// TIA Portal V17 export
// export: Created 2025-03-05T07:59:22.9336726Z, ExportSetting WithDefaults, DisplayName Totally Integrated Automation Portal, DisplayVersion V17 Update 8, DisplayName TIA Portal Openness, DisplayVersion V17 Update 8, DisplayName TIA Portal Version Control Interface, DisplayVersion V17, DisplayName SINAMICS Startdrive Advanced, DisplayVersion V17 SP2, DisplayName SINAMICS Startdrive G110M, G120, G120C, G120D, G120P, G115D, DisplayVersion V17 SP2, DisplayName SINAMICS Startdrive G130, G150, S120, S150, SINAMICS MV, S210, DisplayVersion V17 SP2, DisplayName STEP 7 Professional, DisplayVersion V17 Update 8, DisplayName SINUMERIK ONE STEP 7 Toolbox, DisplayVersion V17 Update 12, DisplayName SINUMERIK 840D sl STEP 7 Toolbox, DisplayVersion V17 Update 12, DisplayName STEP 7 Safety, DisplayVersion V17 Update 6, DisplayName WinCC Advanced, DisplayVersion V17 Update 8
DATA_BLOCK "DB7340_POWDER_PLC_INTERLOCK"   // DB7340
{ S7_Optimized_Access := 'FALSE'; DB_Accessible_From_OPC_UA := 'FALSE' }
AUTHOR : ETXETAR
VERSION : 1.0
// stored: AutoNumber false, DBAccessibleFromOPCUA false, DBAccessibleFromWebserver true, IsOnlyStoredInLoadMemory false, IsWriteProtectedInAS false
   VAR RETAIN
      POWDER_TO_NCU : Struct
         LIFE_BIT : Bool;   // LIFE BIT
         POWDER_UNIT_01_READY_TO_RUN : Bool;   // POWDER UNIT 01 READY TO RUN
         POWDER_UNIT_02_READY_TO_RUN : Bool;   // POWDER UNIT 02 READY TO RUN
         POWDER_UNIT_01_STOPPED : Bool;   // POWDER UNIT 01 STOPPED
         POWDER_UNIT_02_STOPPED : Bool;   // POWDER UNIT 02 STOPPED
         SPARE_05 : Bool;
         SPARE_06 : Bool;
         SPARE_07 : Bool;
         POWDER_PLC_AUTO_MODE : Bool;   // POWDER PLC IN AUTO MODE
         POWDER_PLC_MAN_MODE : Bool;   // POWDER PLC IN MANUAL MODE
         SPARE_12 : Bool;
         SPARE_13 : Bool;
         SPARE_14 : Bool;
         SPARE_15 : Bool;
         SPARE_16 : Bool;
         SPARE_17 : Bool;
         SWITCHED_ON_POWDER_UNIT_01 : Bool;   // SWITCHED ON POWDER UNIT 01
         SWITCHED_ON_POWDER_UNIT_02 : Bool;   // SWITCHED ON POWDER UNIT 02
         SWITCHED_OFF_POWDER_UNIT_01 : Bool;   // SWITCHED OFF POWDER UNIT 01
         SWITCHED_OFF_POWDER_UNIT_02 : Bool;   // SWITCHED OFF POWDER UNIT 02
         SWITCHED_ON_TEMPERATURE_JACKET_UNIT_01 : Bool;   // SWITCHED ON TEMPERATURE JACKET UNIT 01
         SWITCHED_ON_TEMPERATURE_JACKET_UNIT_02 : Bool;   // SWITCHED ON TEMPERATURE JACKET UNIT 02
         SWITCHED_OFF_TEMPERATURE_JACKET_UNIT_01 : Bool;   // SWITCHED OFF TEMPERATURE JACKET UNIT 01
         SWITCHED_OFF_TEMPERATURE_JACKET_UNIT_02 : Bool;   // SWITCHED OFF TEMPERATURE JACKET UNIT 02
         SPARE_30 : Bool;
         SPARE_31 : Bool;
         SPARE_32 : Bool;
         SPARE_33 : Bool;
         SPARE_34 : Bool;
         SPARE_35 : Bool;
         SPARE_36 : Bool;
         SPARE_37 : Bool;
         SPARE_38 : Bool;
         SPARE_39 : Bool;
         SPARE_40 : Bool;
         SPARE_41 : Bool;
         SPARE_44 : Bool;
         SPARE_45 : Bool;
         SPARE_46 : Bool;
         SPARE_47 : Bool;
         POWDER_UNIT_01_ALARM : Bool;   // POWDER UNIT 01 ALARM
         POWDER_UNIT_02_ALARM : Bool;   // POWDER UNIT 02 ALARM
         SPARE_52 : Bool;
         SPARE_53 : Bool;
         SPARE_54 : Bool;
         SPARE_55 : Bool;
         SPARE_56 : Bool;
         SPARE_57 : Bool;
         SPARE_60 : Bool;
         SPARE_61 : Bool;
         SPARE_62 : Bool;
         SPARE_63 : Bool;
         SPARE_64 : Bool;
         SPARE_65 : Bool;
         SPARE_66 : Bool;
         SPARE_67 : Bool;
         SPARE_70 : Bool;
         SPARE_71 : Bool;
         SPARE_72 : Bool;
         SPARE_73 : Bool;
         SPARE_74 : Bool;
         SPARE_75 : Bool;
         SPARE_76 : Bool;
         SPARE_77 : Bool;
         SPARE_80 : Bool;
         SPARE_81 : Bool;
         SPARE_82 : Bool;
         SPARE_83 : Bool;
         SPARE_84 : Bool;
         SPARE_85 : Bool;
         SPARE_86 : Bool;
         SPARE_87 : Bool;
         SPARE_90 : Bool;
         SPARE_91 : Bool;
         SPARE_92 : Bool;
         SPARE_93 : Bool;
         SPARE_94 : Bool;
         SPARE_95 : Bool;
         SPARE_96 : Bool;
         SPARE_97 : Bool;
         UNIT_01_POWDER_FEEDER_1_CARRIER_GAS_ACTUAL_LINE_1 : Real;   // UNIT 01 POWDER FEEDER 1 CARRIER GAS ACTUAL LINE 1
         UNIT_01_POWDER_FEEDER_1_CARRIER_GAS_ACTUAL_LINE_2 : Real;   // UNIT 01 POWDER FEEDER 1 CARRIER GAS ACTUAL LINE 2
         UNIT_01_POWDER_FEEDER_1_DISK_SPEED_ACTUAL_LINE_1 : Real;   // UNIT 01 POWDER FEEDER 1 DISK SPEED ACTUAL LINE 1
         UNIT_01_POWDER_FEEDER_1_DISK_SPEED_ACTUAL_LINE_2 : Real;   // UNIT 01 POWDER FEEDER 1 DISK SPEED ACTUAL LINE 2
         UNIT_01_POWDER_FEEDER_1_STIRRER_SPEED_ACTUAL_LINE_1 : Real;   // UNIT 01 POWDER FEEDER 1 STIRRER SPEED ACTUAL LINE 1
         UNIT_01_POWDER_FEEDER_1_STIRRER_SPEED_ACTUAL_LINE_2 : Real;   // UNIT 01 POWDER FEEDER 1 STIRRER SPEED ACTUAL LINE 2
         UNIT_01_POWDER_FEEDER_1_HOPPER_TEMPERATURE_ACTUAL_LINE_1 : Real;   // UNIT 01 POWDER FEEDER 1 HOPPER TEMPERATURE ACTUAL LINE 1
         UNIT_01_POWDER_FEEDER_1_HOPPER_TEMPERATURE_ACTUAL_LINE_2 : Real;   // UNIT 01 POWDER FEEDER 1 HOPPER TEMPERATURE ACTUAL LINE 2
         UNIT_02_POWDER_FEEDER_1_CARRIER_GAS_ACTUAL_LINE_1 : Real;   // UNIT 02 POWDER FEEDER 1 CARRIER GAS ACTUAL LINE 1
         UNIT_02_POWDER_FEEDER_1_CARRIER_GAS_ACTUAL_LINE_2 : Real;   // UNIT 02 POWDER FEEDER 1 CARRIER GAS ACTUAL LINE 2
         UNIT_02_POWDER_FEEDER_1_DISK_SPEED_ACTUAL_LINE_1 : Real;   // UNIT 02 POWDER FEEDER 1 DISK SPEED ACTUAL LINE 1
         UNIT_02_POWDER_FEEDER_1_DISK_SPEED_ACTUAL_LINE_2 : Real;   // UNIT 02 POWDER FEEDER 1 DISK SPEED ACTUAL LINE 2
         UNIT_02_POWDER_FEEDER_1_STIRRER_SPEED_ACTUAL_LINE_1 : Real;   // UNIT 02 POWDER FEEDER 1 STIRRER SPEED ACTUAL LINE 1
         UNIT_02_POWDER_FEEDER_1_STIRRER_SPEED_ACTUAL_LINE_2 : Real;   // UNIT 02 POWDER FEEDER 1 STIRRER SPEED ACTUAL LINE 2
         UNIT_02_POWDER_FEEDER_1_HOPPER_TEMPERATURE_ACTUAL_LINE_1 : Real;   // UNIT 02 POWDER FEEDER 1 HOPPER TEMPERATURE ACTUAL LINE 1
         UNIT_02_POWDER_FEEDER_1_HOPPER_TEMPERATURE_ACTUAL_LINE_2 : Real;   // UNIT 02 POWDER FEEDER 1 HOPPER TEMPERATURE ACTUAL LINE 2
         UNIT_02_POWDER_FEEDER_2_CARRIER_GAS_ACTUAL_LINE_1 : Real;   // UNIT 02 POWDER FEEDER 2 CARRIER GAS ACTUAL LINE 1
         UNIT_02_POWDER_FEEDER_2_CARRIER_GAS_ACTUAL_LINE_2 : Real;   // UNIT 02 POWDER FEEDER 2 CARRIER GAS ACTUAL LINE 2
         UNIT_02_POWDER_FEEDER_2_DISK_SPEED_ACTUAL_LINE_1 : Real;   // UNIT 02 POWDER FEEDER 2 DISK SPEED ACTUAL LINE 1
         UNIT_02_POWDER_FEEDER_2_DISK_SPEED_ACTUAL_LINE_2 : Real;   // UNIT 02 POWDER FEEDER 2 DISK SPEED ACTUAL LINE 2
         UNIT_02_POWDER_FEEDER_2_STIRRER_SPEED_ACTUAL_LINE_1 : Real;   // UNIT 02 POWDER FEEDER 2 STIRRER SPEED ACTUAL LINE 1
         UNIT_02_POWDER_FEEDER_2_STIRRER_SPEED_ACTUAL_LINE_2 : Real;   // UNIT 02 POWDER FEEDER 2 STIRRER SPEED ACTUAL LINE 2
         UNIT_02_POWDER_FEEDER_2_HOPPER_TEMPERATURE_ACTUAL_LINE_1 : Real;   // UNIT 02 POWDER FEEDER 2 HOPPER TEMPERATURE ACTUAL LINE 1
         UNIT_02_POWDER_FEEDER_2_HOPPER_TEMPERATURE_ACTUAL_LINE_2 : Real;   // UNIT 02 POWDER FEEDER 2 HOPPER TEMPERATURE ACTUAL LINE 2
         SPARE_BYTES : Array[106..199] of Byte;
      END_STRUCT;
      NCU_TO_POWDER : Struct
         LIFE_BIT : Bool;   // LIFE BIT
         PNEUMATIC_SYSTEM_ON : Bool;   // PNEUMATIC SYSTEM ON
         GAS_SYSTEM_ON : Bool;   // GAS SYSTEM ON
         SPARE_04 : Bool;
         SPARE_05 : Bool;
         SPARE_06 : Bool;
         SPARE_07 : Bool;
         LASER_UNIT_01_ACTIVE : Bool;   // LASER UNIT 01 ACTIVE
         LASER_UNIT_02_ACTIVE : Bool;   // LASER UNIT 02 ACTIVE
         ASPIRATION_UNIT_01_OK : Bool;   // ASPIRATION UNIT 01 OK
         ASPIRATION_UNIT_02_OK : Bool;   // ASPIRATION UNIT 02 OK
         U01_PF1_CONDITIONS_OK : Bool;   // UNIT 01 POWDER FEEDER 1 CONDITIONS TO SWITCH ON
         U02_PF1_CONDITIONS_OK : Bool;   // UNIT 02 POWDER FEEDER 1 CONDITIONS TO SWITCH ON
         U02_PF2_CONDITIONS_OK : Bool;   // UNIT 02 POWDER FEEDER 2 CONDITIONS TO SWITCH ON
         SPARE_17 : Bool;
         SWITCH_ON_POWDER_UNIT_01 : Bool;   // SWITCH ON POWDER UNIT 01
         SWITCH_ON_POWDER_UNIT_02 : Bool;   // SWITCH ON POWDER UNIT 02
         SWITCH_OFF_POWDER_UNIT_01 : Bool;   // SWITCH OFF POWDER UNIT 01
         SWITCH_OFF_POWDER_UNIT_02 : Bool;   // SWITCH OFF POWDER UNIT 02
         SWITCH_ON_TEMPERATURE_JACKET_UNIT_01 : Bool;   // SWITCH ON TEMPERATURE JACKET UNIT 01
         SWITCH_ON_TEMPERATURE_JACKET_UNIT_02 : Bool;   // SWITCH ON TEMPERATURE JACKET UNIT 02
         SWITCH_OFF_TEMPERATURE_JACKET_UNIT_01 : Bool;   // SWITCH OFF TEMPERATURE JACKET UNIT 01
         SWITCH_OFF_TEMPERATURE_JACKET_UNIT_02 : Bool;   // SWITCH OFF TEMPERATURE JACKET UNIT 02
         SPARE_30 : Bool;
         SPARE_31 : Bool;
         SPARE_32 : Bool;
         SPARE_33 : Bool;
         SPARE_34 : Bool;
         SPARE_35 : Bool;
         SPARE_36 : Bool;
         SPARE_37 : Bool;
         SELECT_ARGON_GAS : Bool;   // SELECT ARGON GAS
         SELECT_NITROGEN_GAS : Bool;   // SELECT NITROGEN GAS
         SELECT_IMPERIAL_SYSTEM : Bool;   // SELECT IMPERIAL SYSTEM
         SELECT_METRIC_SYSTEM : Bool;   // SELECT METRIC SYSTEM
         SPARE_44 : Bool;
         SPARE_45 : Bool;
         SPARE_46 : Bool;
         SPARE_47 : Bool;
         LASER_MEDICOAT_UNIT_01_ALARM : Bool;   // LASER MEDICOAT UNIT 01 ALARM
         LASER_MEDICOAT_UNIT_02_ALARM : Bool;   // LASER MEDICOAT UNIT 02 ALARM
         SPARE_52 : Bool;
         SPARE_53 : Bool;
         SPARE_54 : Bool;
         SPARE_55 : Bool;
         SPARE_56 : Bool;
         SPARE_57 : Bool;
         SPARE_60 : Bool;
         SPARE_61 : Bool;
         SPARE_62 : Bool;
         SPARE_63 : Bool;
         SPARE_64 : Bool;
         SPARE_65 : Bool;
         SPARE_66 : Bool;
         SPARE_67 : Bool;
         SPARE_70 : Bool;
         SPARE_71 : Bool;
         SPARE_72 : Bool;
         SPARE_73 : Bool;
         SPARE_74 : Bool;
         SPARE_75 : Bool;
         SPARE_76 : Bool;
         SPARE_77 : Bool;
         SPARE_80 : Bool;
         SPARE_81 : Bool;
         SPARE_82 : Bool;
         SPARE_83 : Bool;
         SPARE_84 : Bool;
         SPARE_85 : Bool;
         SPARE_86 : Bool;
         SPARE_87 : Bool;
         SPARE_90 : Bool;
         SPARE_91 : Bool;
         SPARE_92 : Bool;
         SPARE_93 : Bool;
         SPARE_94 : Bool;
         SPARE_95 : Bool;
         SPARE_96 : Bool;
         SPARE_97 : Bool;
         UNIT_01_POWDER_FEEDER_1_CARRIER_GAS_NOMINAL_LINE_1 : Real;   // UNIT 01 POWDER FEEDER 1 CARRIER GAS NOMINAL LINE 1
         UNIT_01_POWDER_FEEDER_1_CARRIER_GAS_NOMINAL_LINE_2 : Real;   // UNIT 01 POWDER FEEDER 1 CARRIER GAS NOMINAL LINE 2
         UNIT_01_POWDER_FEEDER_1_DISK_SPEED_NOMINAL_LINE_1 : Real;   // UNIT 01 POWDER FEEDER 1 DISK SPEED NOMINAL LINE 1
         UNIT_01_POWDER_FEEDER_1_DISK_SPEED_NOMINAL_LINE_2 : Real;   // UNIT 01 POWDER FEEDER 1 DISK SPEED NOMINAL LINE 2
         UNIT_01_POWDER_FEEDER_1_STIRRER_SPEED_NOMINAL_LINE_1 : Real;   // UNIT 01 POWDER FEEDER 1 STIRRER SPEED NOMINAL LINE 1
         UNIT_01_POWDER_FEEDER_1_STIRRER_SPEED_NOMINAL_LINE_2 : Real;   // UNIT 01 POWDER FEEDER 1 STIRRER SPEED NOMINAL LINE 2
         UNIT_01_POWDER_FEEDER_1_HOPPER_TEMPERATURE_NOMINAL_LINE_1 : Real;   // UNIT 01 POWDER FEEDER 1 HOPPER TEMPERATURE NOMINAL LINE 1
         UNIT_01_POWDER_FEEDER_1_HOPPER_TEMPERATURE_NOMINAL_LINE_2 : Real;   // UNIT 01 POWDER FEEDER 1 HOPPER TEMPERATURE NOMINAL LINE 2
         UNIT_02_POWDER_FEEDER_1_CARRIER_GAS_NOMINAL_LINE_1 : Real;   // UNIT 02 POWDER FEEDER 1 CARRIER GAS NOMINAL LINE 1
         UNIT_02_POWDER_FEEDER_1_CARRIER_GAS_NOMINAL_LINE_2 : Real;   // UNIT 02 POWDER FEEDER 1 CARRIER GAS NOMINAL LINE 2
         UNIT_02_POWDER_FEEDER_1_DISK_SPEED_NOMINAL_LINE_1 : Real;   // UNIT 02 POWDER FEEDER 1 DISK SPEED NOMINAL LINE 1
         UNIT_02_POWDER_FEEDER_1_DISK_SPEED_NOMINAL_LINE_2 : Real;   // UNIT 02 POWDER FEEDER 1 DISK SPEED NOMINAL LINE 2
         UNIT_02_POWDER_FEEDER_1_STIRRER_SPEED_NOMINAL_LINE_1 : Real;   // UNIT 02 POWDER FEEDER 1 STIRRER SPEED NOMINAL LINE 1
         UNIT_02_POWDER_FEEDER_1_STIRRER_SPEED_NOMINAL_LINE_2 : Real;   // UNIT 02 POWDER FEEDER 1 STIRRER SPEED NOMINAL LINE 2
         UNIT_02_POWDER_FEEDER_1_HOPPER_TEMPERATURE_NOMINAL_LINE_1 : Real;   // UNIT 02 POWDER FEEDER 1 HOPPER TEMPERATURE NOMINAL LINE 1
         UNIT_02_POWDER_FEEDER_1_HOPPER_TEMPERATURE_NOMINAL_LINE_2 : Real;   // UNIT 02 POWDER FEEDER 1 HOPPER TEMPERATURE NOMINAL LINE 2
         UNIT_02_POWDER_FEEDER_2_CARRIER_GAS_NOMINAL_LINE_1 : Real;   // UNIT 02 POWDER FEEDER 2 CARRIER GAS NOMINAL LINE 1
         UNIT_02_POWDER_FEEDER_2_CARRIER_GAS_NOMINAL_LINE_2 : Real;   // UNIT 02 POWDER FEEDER 2 CARRIER GAS NOMINAL LINE 2
         UNIT_02_POWDER_FEEDER_2_DISK_SPEED_NOMINAL_LINE_1 : Real;   // UNIT 02 POWDER FEEDER 2 DISK SPEED NOMINAL LINE 1
         UNIT_02_POWDER_FEEDER_2_DISK_SPEED_NOMINAL_LINE_2 : Real;   // UNIT 02 POWDER FEEDER 2 DISK SPEED NOMINAL LINE 2
         UNIT_02_POWDER_FEEDER_2_STIRRER_SPEED_NOMINAL_LINE_1 : Real;   // UNIT 02 POWDER FEEDER 2 STIRRER SPEED NOMINAL LINE 1
         UNIT_02_POWDER_FEEDER_2_STIRRER_SPEED_NOMINAL_LINE_2 : Real;   // UNIT 02 POWDER FEEDER 2 STIRRER SPEED NOMINAL LINE 2
         UNIT_02_POWDER_FEEDER_2_HOPPER_TEMPERATURE_NOMINAL_LINE_1 : Real;   // UNIT 02 POWDER FEEDER 2 HOPPER TEMPERATURE NOMINAL LINE 1
         UNIT_02_POWDER_FEEDER_2_HOPPER_TEMPERATURE_NOMINAL_LINE_2 : Real;   // UNIT 02 POWDER FEEDER 2 HOPPER TEMPERATURE NOMINAL LINE 2
         SPARE_BYTES_106 : Array[106..129] of Byte;
         CURRENT_PROTECTION_LEVEL : Byte;   // CURRENT ACCESS LEVEL
         EKS_IDENT_1 : Byte;   // EKS OPERATOR ID CHAR 1
         EKS_IDENT_2 : Byte;   // EKS OPERATOR ID CHAR 2
         EKS_IDENT_3 : Byte;   // EKS OPERATOR ID CHAR 3
         EKS_IDENT_4 : Byte;   // EKS OPERATOR ID CHAR 4
         EKS_IDENT_5 : Byte;   // EKS OPERATOR ID CHAR 5
         EKS_IDENT_6 : Byte;   // EKS OPERATOR ID CHAR 6
         EKS_IDENT_7 : Byte;   // EKS OPERATOR ID CHAR 7
         EKS_OPERATOR_IDENTIFICATION : Byte;
         EKS_IDENT_8 : Byte;
         SPARE_BYTES_140 : Array[140..199] of Byte;
      END_STRUCT;
   END_VAR
BEGIN
END_DATA_BLOCK
